// TIA Portal V17 export
// export: Created 2023-06-23T18:33:37.5603751Z, ExportSetting WithDefaults, DisplayName Totally Integrated Automation Portal, DisplayVersion V17, DisplayName TIA Portal Openness, DisplayVersion V17, DisplayName TIA Portal Version Control Interface, DisplayVersion V17, DisplayName STEP 7 Professional, DisplayVersion V17, DisplayName STEP 7 Safety, DisplayVersion V17, DisplayName WinCC Advanced / Unified PC, DisplayVersion V17
VAR_GLOBAL   // PLC tag table "04_EL-4"
   "iEL-4p" AT %I1.0 : Bool;
   "iEL-4" AT %I1.1 : Bool;
   "oEL-4p" AT %Q0.2 : Bool;
   "oEL-4" AT %Q0.3 : Bool;
END_VAR
